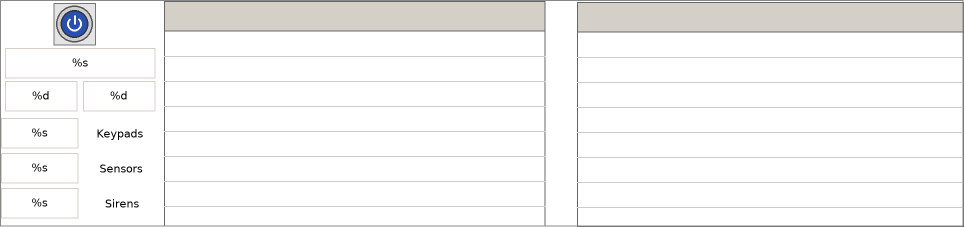
VISUALIZATION Alarm  // 964x227
VAR_IN_OUT
	stAlarm		: ST_AlarmManagerHMI;
END_VAR
    PowerSwitch (50,3 49x42), variable: stAlarm.eState = E_AlarmState.Enabled, input disabled if: TRUE, behaviour: TOGGLE, style: Switch-PowerSwitch-Blue
    Table (164,1 381x225), data array: stAlarm.aSensors
        p3854506369: stAlarm.aSensors[INDEX].sName
        p1892666644: stAlarm.aSensors[INDEX].nID
        p338671338: stAlarm.aSensors[INDEX].bAlarm
        p2170511999: stAlarm.aSensors[INDEX].bTamper
    Table (577,2 387x225), data array: stAlarm.aSirens
        p3854506369: stAlarm.aSirens[INDEX].sName
        p1892666644: stAlarm.aSirens[INDEX].nID
        p338671338: stAlarm.aSirens[INDEX].bSiren
        p2170511999: stAlarm.aSirens[INDEX].bLight
        p3723444502: stAlarm.aSirens[INDEX].bTamper
    Textfield (1,118 77x30), "%s", text variable: stAlarm.nKeypads
    Textfield (1,153 77x30), "%s", text variable: stAlarm.nSensors
    Textfield (1,188 77x30), "%s", text variable: stAlarm.nSirens
    Label (85,119 70x30), "Keypads"
    Label (86,154 70x30), "Sensors"
    Label (87,189 70x30), "Sirens"
    Textfield (5,48 150x30), "%s", text variable: stAlarm.eState
    Textfield (5,81 72x30), "%d", text variable: stAlarm.nActiveID
    Textfield (83,81 72x30), "%d", text variable: stAlarm.nActiveReason
END_VISUALIZATION

(* stored: Version 1.1.0.1, ProductVersion 3.1.4024.12
   Visu Alarm: Id {1701f66b-e5a7-4a0b-b7c2-bac8982c9206} *)
